FUNCTION_BLOCK FB_DigitalOutput EXTENDS FB_ComponentBase
VAR
	/// IO reference
	stOut 					: REFERENCE TO ST_DigitalOutputOut;
	
	fbButton				: FB_sensor;
	
	fbSignal				: FB_TON_RMTH;
	
	tDelay					: TIME;
	
END_VAR

METHOD AutoOff
VAR_INPUT
	Delay					: TIME;
END_VAR
tDelay:= Delay;
END_METHOD

METHOD FB_init : BOOL
VAR_INPUT
	bInitRetains : BOOL; // if TRUE, the retain variables are initialized (warm start / cold start)
	bInCopyCode : BOOL;  // if TRUE, the instance afterwards gets moved into the copy code (online change)
END_VAR
eTyp := E_ComponentType.eComponentType_DigitalOutput;
END_METHOD

PROPERTY OutputState : BOOL
GET
OutputState := stOut.bOutput;
END_GET
END_PROPERTY

METHOD Reset
VAR_INPUT
END_VAR
// base logic run
SUPER^.Reset();

IF NOT __ISVALIDREF(stOut) THEN
	RETURN;
END_IF

stOut.bOutput := FALSE;
END_METHOD

/// Run component logic
{attribute 'object_name' := 'Run'}
METHOD Run : E_ComponentState
VAR_INPUT
END_VAR
// base logic run
Run := SUPER^.Run();

IF NOT __ISVALIDREF(stOut) THEN
	RETURN;
END_IF

fbSignal(in:= stOut.bOutput, pt:=tDelay);

// auto switch off
IF tDelay <> T#0S AND fbSignal.Q THEN
	stOut.bOutput := FALSE;
END_IF
END_METHOD

METHOD SetReferences : E_OperationResult
VAR_IN_OUT
	/// IO structure
	DigitalOutput 		: ST_DigitalOutputIO;
END_VAR
stOut REF= DigitalOutput.stOut;
END_METHOD

METHOD SwitchState
VAR_INPUT
	bEnable				: BOOL;
END_VAR
stout.bOutput := bEnable;
END_METHOD

END_FUNCTION_BLOCK

(* stored: Version 1.1.0.1, ProductVersion 3.1.4022.10
   POU FB_DigitalOutput: Id {7a1b4279-643f-4dd3-b476-66c65e5d5c14}, SpecialFunc None
   Folder Factory: Id {8f45a723-4b92-4443-905b-54356b390988}
   Folder Properties: Id {e3c546d1-1da3-4093-a99f-46a1641ca42d}
   Method AutoOff: Id {32887618-f119-42cc-89c7-266c605cafd9}
   Method FB_init: Id {ce813b69-a7e0-459d-b586-c372a8b01927}
   Property OutputState: Id {9e3bf72a-dc3e-48d6-abea-70df58e7c678}
   Get Get: Id {d58b873f-5096-4ced-96c5-783090248851}
   Method Reset: Id {8bb56281-5db6-49b1-a74d-b8976b878f5d}
   Method Run: Id {7794ab06-27f2-40a1-81ef-128c9449c925}
   Method SetReferences: Id {6c69d759-090d-462e-945b-b4fde1a7b9b7}
   Method SwitchState: Id {a8c46daa-6b51-4378-bfa7-3acaf30e0fac} *)
